INTERFACE I_DeserializerFeedbackVisitor EXTENDS I_ErrorVisitor

METHOD VisitDeserializerFeedback
VAR_INPUT
	VisitingDeserializerFeedback : I_DeserializerFeedback;
END_VAR
END_METHOD

END_INTERFACE

(* stored: Version 1.1.0.1, ProductVersion 3.1.4024.12
   Itf I_DeserializerFeedbackVisitor: Id {f975dca1-7260-03bc-219b-f3b54a16abc6}
   Method VisitDeserializerFeedback: Id {456b92fc-0237-4201-a084-5cd05bdb1c89} *)
